FUNCTION TryConvert_USINT_TO_ULINT : BOOL
VAR_INPUT
	in : USINT;
	out : REFERENCE TO ULINT;
END_VAR

out := USINT_TO_ULINT(in);
TryConvert_USINT_TO_ULINT := TRUE;

END_FUNCTION

(* stored: Version 1.1.0.1, ProductVersion 3.1.4024.12
   POU TryConvert_USINT_TO_ULINT: Id {1fa759a8-a825-4983-868f-36f5894fc43c}, SpecialFunc None *)
